Universal Robots PolyScope program: xiaomi.urp

Program xiaomi (installation=20240827 directory=/programs/Demos/adaptiveGrip/新文件夹 createdIn=5.15.1 lastSavedIn=5.15.1 robotSerialNumber=20245500285)
Calibrated DH parameters: a=[0.000097, -0.210459, -0.026602, 0.000137, 0.000078, 0]; d=[0.162601, 254.180657, -54.076236, -199.970743, 0.099615, 0.099684]; alpha=[1.569796, -0.001455, 0.001957, 1.570525, -1.571561, 0]; deltaTheta=[0, -1.053331, 8.839472, -1.50296, 0.000002, 0]
InitVariablesNode
BeforeStart
  SuppressedNode
    MoveL speed 250 mm/s, acceleration 1200 mm/s^2 (useActiveTCP=true) feature=Base
      Waypoint ppick: TCP in base x=-36.634 y=-638.502 z=14.663 mm, rx=2.1795 ry=2.2626 rz=-0.0001 rad; joints [74.558, -61.012, 96.454, -125.49, -90.074, 72.599] deg; TCP offset x=-0.17 y=0 z=192.95 mm, rx=0 ry=0 rz=0 rad
      Waypoint pappro: TCP in base x=-36.657 y=-638.51 z=49.536 mm, rx=2.1795 ry=2.2625 rz=-0.0002 rad; joints [74.558, -63.595, 94.504, -120.959, -90.063, 72.602] deg
  Script: usb = rpc_factory("xmlrpc","http://192.168.1.7:9120/RPC2")
  Script: usb.open()
Robot Program (runOnlyOnce=false)
  Placeholder
